// TwinCAT 3 PLC project main
// ProgramVersion: 3.1.4024.0
// libraries:
//   Tc2_Standard, * (Beckhoff Automation GmbH)
//   Tc2_System, * (Beckhoff Automation GmbH)
//   Tc3_Module, * (Beckhoff Automation GmbH)
// project tree:
//   / GlobalTextList.TcGTLO, PlcTask.TcTTO, Visualization Manager.TcVMO (not stored)
//   POUs/ MAIN.TcPOU
//   VISUs/ Visu.TcVIS
// real-time tasks:
//   TASK PlcTask: cycle T#10ms, priority 20, ADS port 350

CONFIGURATION main
    RESOURCE PLC ON TwinCAT3
        TASK PlcTask(INTERVAL := T#10ms, PRIORITY := 20);
        PROGRAM MAIN WITH PlcTask : MAIN;
    END_RESOURCE
END_CONFIGURATION

// ---- POUs/MAIN.TcPOU
PROGRAM MAIN
VAR
	b_groen_h 	: BOOL;
	b_oranje_h 	: BOOL;
	b_rood_h 	: BOOL;
	b_rood_v 	: BOOL;
	b_groen_v 	: BOOL;
	b_oranje_v 	: BOOL;
END_VAR

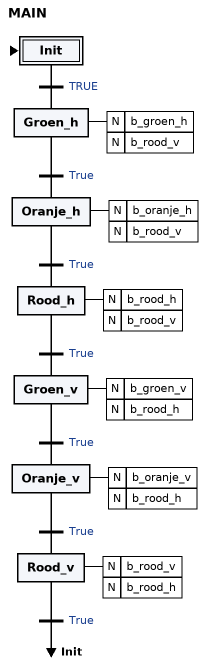
INITIAL_STEP Init:
END_STEP
TRANSITION FROM Init TO Groen_h
    := TRUE;
END_TRANSITION
STEP Groen_h:  // min time t#1000ms
    b_groen_h(N);
    b_rood_v(N);
END_STEP
TRANSITION FROM Groen_h TO Oranje_h
    := True;
END_TRANSITION
STEP Oranje_h:  // min time t#1000ms
    b_oranje_h(N);
    b_rood_v(N);
END_STEP
TRANSITION FROM Oranje_h TO Rood_h
    := True;
END_TRANSITION
STEP Rood_h:  // min time t#1000ms
    b_rood_h(N);
    b_rood_v(N);
END_STEP
TRANSITION FROM Rood_h TO Groen_v
    := True;
END_TRANSITION
STEP Groen_v:  // min time t#1000ms
    b_groen_v(N);
    b_rood_h(N);
END_STEP
TRANSITION FROM Groen_v TO Oranje_v
    := True;
END_TRANSITION
STEP Oranje_v:  // min time t#1000ms
    b_oranje_v(N);
    b_rood_h(N);
END_STEP
TRANSITION FROM Oranje_v TO Rood_v
    := True;
END_TRANSITION
STEP Rood_v:  // min time t#1000ms
    b_rood_v(N);
    b_rood_h(N);
END_STEP
TRANSITION FROM Rood_v TO Init
    := True;
END_TRANSITION

END_PROGRAM

// ---- VISUs/Visu.TcVIS
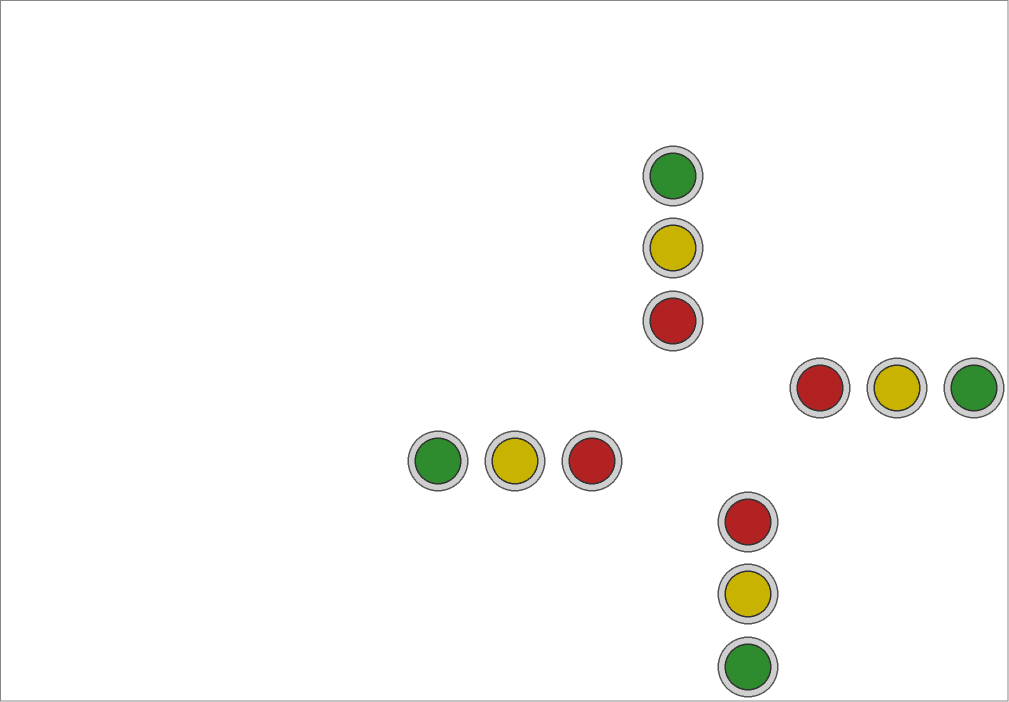
VISUALIZATION Visu  // 1009x702
    Group (403,426 224x70)
        Lamp1 (154,0 70x70), variable: MAIN.b_rood_h, style: Lamp-Lamp1-Red
        Lamp1 (77,0 70x70), variable: MAIN.b_oranje_h, style: Lamp-Lamp1-Yellow
        Lamp1 (0,0 70x70), variable: MAIN.b_groen_h, style: Lamp-Lamp1-Green
    Group (785,353 224x70)
        Lamp1 (154,0 70x70), variable: MAIN.b_groen_h, style: Lamp-Lamp1-Green
        Lamp1 (77,0 70x70), variable: MAIN.b_oranje_h, style: Lamp-Lamp1-Yellow
        Lamp1 (0,0 70x70), variable: MAIN.b_rood_h, style: Lamp-Lamp1-Red
    Group (713,487 70x215)
        Lamp1 (0,0 70x70), variable: MAIN.b_rood_v, style: Lamp-Lamp1-Red
        Lamp1 (0,72 70x70), variable: MAIN.b_oranje_v, style: Lamp-Lamp1-Yellow
        Lamp1 (0,145 70x70), variable: MAIN.b_groen_v, style: Lamp-Lamp1-Green
    Group (638,141 70x215)
        Lamp1 (0,0 70x70), variable: MAIN.b_groen_v, style: Lamp-Lamp1-Green
        Lamp1 (0,72 70x70), variable: MAIN.b_oranje_v, style: Lamp-Lamp1-Yellow
        Lamp1 (0,145 70x70), variable: MAIN.b_rood_v, style: Lamp-Lamp1-Red
END_VISUALIZATION
